PROGRAM MAIN
VAR
END_VAR

END_PROGRAM

(* stored: Version 1.1.0.1
   POU MAIN: Id {3e98b677-9ccf-40dc-8818-1c520a2e5252} *)
